# EPICS substitutions: opcua-IOC-demoApp/Db/uasdk-server.substitutions
file "opcuaServerInfo.template" {
pattern { P, R, SESS }
{ "$(PREF)", "$(REC=)", "$(SESSION)" }
}

file "opcuaServerStats.template" {
pattern { P, R, SESS, SUBS }
{ "$(PREF)", "$(REC=)", "$(SESSION)", "$(SUBSCRIPT)" }
}
